TYPE teSimAxisNames :
(
	CE_SIM_AXIS_X:=1,			// X-axis drive
	CE_SIM_AXIS_Y,				// Y-axis drive
	CE_SIM_AXIS_Z,				// Z-axis drive
	CE_SIM_AXIS_C 				// C-axis drive
);
END_TYPE

(* stored: Version 1.1.0.1, ProductVersion 3.1.4022.18
   DUT teSimAxisNames: Id {3c2b48a3-9834-472b-96c0-cd9b533176f2} *)
